FUNCTION_BLOCK FB_CylinderCutY EXTENDS FB_ComponentBase IMPLEMENTS I_Cylinder
VAR
    // Internal variables
    _ExtendRequestY  : BOOL;
    _RetractRequestY : BOOL;
    _ExtendedY       : BOOL;
    _RetractedY      : BOOL;
    _ExtendingY      : BOOL;
    _RetractingY     : BOOL;


    Extend_RTRIG  : R_TRIG;
    Retract_RTRIG : R_TRIG;

    //HMI 
    Cylinder_HMI : ST_Cylinder_HMI;
	
	// Timery ruchu
    MovementTimer : TON;
    
    // Alarmy
    CylinderAlarms : ARRAY[1..3] OF FB_TcAlarm;
END_VAR

VAR_INPUT
   	CylinderSensorCutY 			AT%I*		:	BOOL;
END_VAR

VAR_OUTPUT
	CylinderValveCutY			AT%Q*		:	BOOL;
END_VAR

PROPERTY Config : ST_Cylinder_Config
GET
Config := Cylinder_HMI.Config;
END_GET
SET
Cylinder_HMI.Config := Config;
END_SET
END_PROPERTY

METHOD PROTECTED CreateEvents
VAR_INPUT
END_VAR
SUPER^.CreateEvents();

// Powiązanie tablicy alarmów z klasą CylinderAlarms z TMC
F_CreateAllEventsInClass(
    Alarms     := CylinderAlarms,
    ClassSize  := SIZEOF(TC_EVENTS.CylinderAlarms),
    pInitEvent := ADR(TC_EVENTS.CylinderAlarms.InitReferenceEvent),
    Prefix     := _Name
);
END_METHOD

METHOD CyclicLogic
// One shot the requests
Extend_RTRIG(CLK := _ExtendRequestY);
Retract_RTRIG(CLK := _RetractRequestY);

// Handle Extend
IF Extend_RTRIG.Q THEN
    CylinderValveCutY := TRUE;
    _ExtendingY       := TRUE;
    _RetractingY      := FALSE;
    _RetractedY       := FALSE;
    _RetractRequestY  := FALSE;
END_IF

// Handle Retract
IF Retract_RTRIG.Q THEN
    CylinderValveCutY := FALSE;
    _ExtendingY       := FALSE;
    _RetractingY      := TRUE;
    _ExtendedY        := FALSE;
    _ExtendRequestY   := FALSE;
END_IF

// Aktualizacja stanu wyłącznie z czujnika
_ExtendedY  := CylinderSensorCutY;
_RetractedY := NOT CylinderSensorCutY;

// Status ruchu – tylko gdy trwa przejście
_ExtendingY  := _ExtendingY  AND NOT _ExtendedY;
_RetractingY := _RetractingY AND NOT _RetractedY;

// Odmierzanie czasu ruchu (używamy SEL żeby brać czas wysuwu lub chowania)
MovementTimer(
    IN := _ExtendingY OR _RetractingY,
    PT := LREAL_TO_TIME(SEL(_ExtendingY, Cylinder_HMI.Config.RetractTimeY, Cylinder_HMI.Config.ExtendTimeY) * 1000.0) 
);

// Wywołanie logiki bazowej komponentu (Tylko raz!)
SUPER^.CyclicLogic();

// Aktualizacja najwyższego priorytetu błędu dla komponentu
_CurrentAlarmSeverity := F_GetMaxSeverityRaised(Alarms := CylinderAlarms, CurrentSeverity := _CurrentAlarmSeverity);
END_METHOD

PROPERTY Error : BOOL
GET
Error := _Error;
END_GET
SET
_Error := Error;
END_SET
END_PROPERTY

METHOD Extend
_ExtendRequestY  := TRUE;
_RetractRequestY := FALSE;
END_METHOD

PROPERTY Extended : BOOL
GET
Extended := _ExtendedY;
END_GET
END_PROPERTY

METHOD PROTECTED HMICommunication
VAR_INPUT
END_VAR
SUPER^.HMICommunication();

//Handle the requests to extend and retract
IF ComponentBase_HMI.Status.HMIControlAvailable THEN
    IF Cylinder_HMI.Command.RetractExtendY THEN
        Extend();
    ELSIF Cylinder_HMI.Command.RetractCylinderY THEN
        Retract();
    END_IF
END_IF

//Update HMI status info
Cylinder_HMI.Status.ExtendedY    := _ExtendedY;
Cylinder_HMI.Status.ExtendingY   := _ExtendingY;
Cylinder_HMI.Status.RetractedY  := _RetractedY;
Cylinder_HMI.Status.RetractingY  := _RetractingY;
END_METHOD

//! @summary Basic component initialization logic
METHOD PROTECTED Initialize : BOOL;

//! @description This method is called by <c>CyclicLogic()</c> as required

IF CylinderSensorCutY THEN
    _ExtendedY  := TRUE;
    _RetractedY := FALSE;
ELSE
    _ExtendedY  := FALSE;
    _RetractedY := TRUE;
END_IF

_ExtendingY      := FALSE;
_ExtendRequestY  := FALSE;
_RetractingY     := FALSE;
_RetractRequestY := FALSE;

Initialize := SUPER^.Initialize();
END_METHOD

METHOD PROTECTED Monitoring
VAR_INPUT
END_VAR
_Busy := _ExtendingY OR _RetractingY;

// Jeśli czas minął, zgłoś odpowiedni błąd
IF MovementTimer.Q THEN
    _Error   := TRUE;
    _ErrorID := 1; 

    IF _ExtendingY AND NOT CylinderAlarms[E_CylinderAlarms.ExtendTimeout].bRaised THEN
        RaiseAlarmWithStrings(CylinderAlarms[E_CylinderAlarms.ExtendTimeout], '', '');
    
    ELSIF _RetractingY AND NOT CylinderAlarms[E_CylinderAlarms.RetractTimeout].bRaised THEN
        RaiseAlarmWithStrings(CylinderAlarms[E_CylinderAlarms.RetractTimeout], '', '');
    END_IF
END_IF

// Resetowanie błędu, gdy cylinder dotrze do celu
IF (_ExtendedY AND _ExtendRequestY) OR (_RetractedY AND _RetractRequestY) THEN
    _Error   := FALSE;
    _ErrorID := 0;
END_IF

SUPER^.Monitoring();
END_METHOD

METHOD Retract
_ExtendRequestY  := FALSE;
_RetractRequestY := TRUE;
END_METHOD

PROPERTY Retracted : BOOL
GET
Retracted := _RetractedY;
END_GET
END_PROPERTY

END_FUNCTION_BLOCK

(* stored: Version 1.1.0.1, ProductVersion 3.1.4024.15
   POU FB_CylinderCutY: Id {8ada12fc-8440-0750-128a-e06d4a970561}, SpecialFunc None
   Folder I_ComponentBase: Id {e725d5a4-2c2c-07e9-2a68-0cf7a1a118b8}
   Folder I_CyclicFB: Id {89d6c8b5-777b-05c8-0d3b-cb03ad048b76}
   Folder I_Cylinder: Id {a88ec890-cbf6-05f6-1fe3-43518715a1a1}
   Property Config: Id {92518cf8-c680-4c31-a6cf-f7fe6fced64c}
   Get Get: Id {49570b44-2aca-4cfd-907b-bfeaaa94c4c0}
   Set Set: Id {b3e9847b-3673-4362-b839-1e77672cdcdf}
   Method CreateEvents: Id {307e5521-2f56-0737-2771-0304ac08c314}
   Method CyclicLogic: Id {523e51c2-13b6-03e9-1aa1-a3c583ef5375}
   Property Error: Id {fa35be3d-1304-4f63-a352-60e04b585c4a}
   Get Get: Id {3d446071-592e-4490-ba75-42df150223c8}
   Set Set: Id {875a67df-099d-4c1f-9198-4b57908183d0}
   Method Extend: Id {f94e6f21-1340-0909-053a-ec233f6345e3}
   Property Extended: Id {05467c14-4f1d-0771-125d-3762d6da92b0}
   Get Get: Id {0a44f002-4454-0333-267c-974316a02102}
   Method HMICommunication: Id {e2d15e2d-6459-0f6b-15c7-82b21fb452fa}
   Method Initialize: Id {89ccf394-b5d3-056c-10fd-042199230882}
   Method Monitoring: Id {9666f76e-680f-0ae2-0499-28e8d172221c}
   Method Retract: Id {6cd1b03b-982c-02c0-0f22-afaa5838a082}
   Property Retracted: Id {636006d7-169f-036d-3ce3-fa2a088901a3}
   Get Get: Id {c67dbb29-58ad-0355-0bc6-42672ce042f9} *)
